Yaskawa INFORM job: VELOCITY_TEST.JBI

/JOB
//NAME VELOCITY_TEST
//POS
///NPOS 7,0,0,0,0,0
///TOOL 5
///POSTYPE PULSE
///PULSE
C00000=-1,-50477,-58433,3,-74929,486
C00001=-9597,18619,-45513,-2349,-31863,4376
C00002=-9596,18619,-45513,-2350,-31865,4376
C00003=-7102,18316,-45929,-1744,-31761,3362
C00004=-6886,21378,-41660,-1661,-32392,3257
C00005=-6886,21378,-41660,-1662,-32393,3259
C00006=-2,-50477,-58433,3,-74939,487
//INST
///DATE 2024/03/04 13:03
///ATTR SC,RW
///GROUP1 RB1
NOP
COMM MOVJ C00000 VJ=5.00
COMM MOVJ C00001 VJ=5.00
MOVL C00002 V=20.0
MOVL C00003 V=20.0
MOVL C00004 V=20.0
MOVL C00005 V=20.0
COMM MOVJ C00006 VJ=5.00
END
